Yaskawa INFORM job: SR-ARC-1.JBI

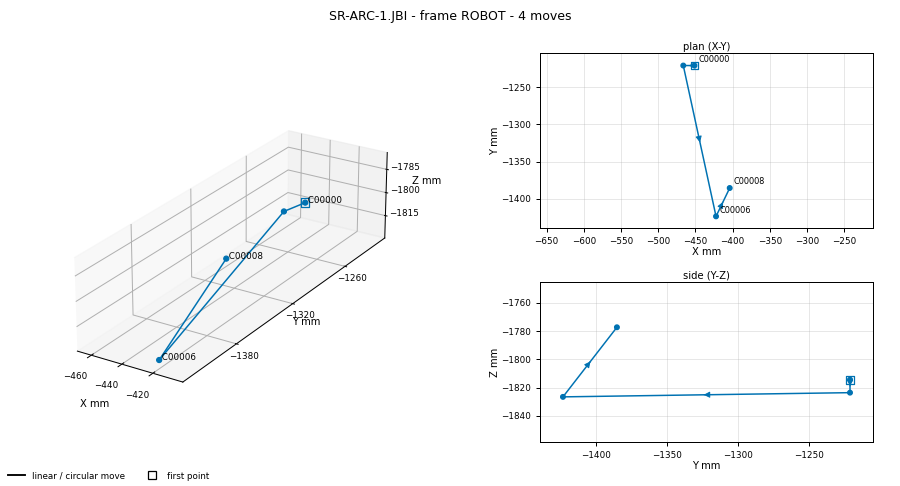
[picture p0: tool path of SR-ARC-1.JBI in frame ROBOT, 4 of 4 moves have a stored position in this frame; points joined in program order, loops and branches not executed]
/JOB
//NAME SR-ARC-1
///FOLDERNAME INNE
//POS
///NPOS 9,6,0,1,0,0
///TOOL 0
///POSTYPE ROBOT
///RECTAN
///RCONF 1,0,0,0,0,0,0,0,0,0,0,0,0,0,0,0,0,0,0,0,0,0,0,0
C00000=-451.283,-1220.754,-1814.351,-40.3761,0.3788,-83.7631
C00001=-466.319,-1220.777,-1823.558,-40.3761,0.3785,-83.7627
///RCONF 0,0,0,0,0,0,0,0,0,0,0,0,0,0,0,0,0,0,0,0,0,0,0,0
C00002=-59.528,-233.360,-1706.636,-45.1397,6.9495,-80.8801
C00003=-59.510,-82.151,-1706.659,-45.1369,6.9489,-80.8804
C00004=-59.526,-233.358,-1706.634,-45.1397,6.9491,-80.8808
///RCONF 1,0,0,0,0,0,0,0,0,0,0,0,0,0,0,0,0,0,0,0,0,0,0,0
C00005=-466.319,-1220.777,-1823.558,-40.3761,0.3785,-83.7627
C00006=-422.293,-1423.586,-1826.532,-40.3759,0.3782,-83.7677
///RCONF 0,0,0,0,0,0,0,0,0,0,0,0,0,0,0,0,0,0,0,0,0,0,0,0
C00007=-56.576,-232.968,-1706.050,-45.0935,7.2921,-80.5361
///RCONF 1,0,0,0,0,0,0,0,0,0,0,0,0,0,0,0,0,0,0,0,0,0,0,0
C00008=-403.896,-1385.468,-1777.357,-40.3747,0.3771,-83.7688
///RCONF 0,0,0,0,0,0,0,0,0,0,0,0,0,0,0,0,0,0,0,0,0,0,0,0
BC00000=2343.226,229.569,1032.178
BC00001=2343.226,229.569,1032.178
BC00002=2343.226,229.569,1032.178
BC00003=2343.226,229.569,1032.178
BC00004=1843.422,4161.120,598.982
BC00005=2343.226,229.569,1032.178
///POSTYPE BASE
P00070=0.003,2.805,-1.116,0.0000,0.0000,0.0000
//INST
///DATE 2023/11/01 18:40
///ATTR SC,RW,RJ
////FRAME ROBOT
///GROUP1 RB1,BS1
NOP
MOVL C00000 BC00000 V=150.0
MOVL C00001 BC00001 V=75.0
COMM MACRO1 MJ#(7) ARGFB000 ARGF1 ARGFC00002 ARGFC00003 ARGF1 ARGF70 ARGF4021 ARGF120 ARGF70
COMM PAUSE IF B001=0
COMM MACRO1 MJ#(8) ARGFB000 ARGFP070 ARGFC00004 ARGF1 ARGF50.0 ARGF71 ARGF4020
COMM PAUSE IF B001=0
COMM ARCON
MACRO1 MJ#(5) ARGFB000 ARGF1 ARGF450 ARGFC00005 ARGFBC00002 ARGF4020
MOVL C00006 BC00003 V=16.7
COMM MACRO1 MJ#(9) ARGFB000 ARGF1
COMM MOVL C00007 BC00004 V=16.7
MACRO1 MJ#(3) ARGFB000
SFTOF
COMM ARCOF
MOVL C00008 BC00005 V=75.0
END
